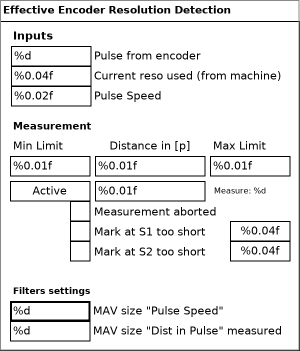
VISUALIZATION _VISU_EffectiveEncoderResolutionDetection  // 300x351
VAR_IN_OUT
	mInst : FB_EffectiveEncoderResolutionDetection;
END_VAR
    Rectangle (0,21 300x330)
    Rectangle (10,116 80x20), "Measurement"
    RoundedRectangle (10,181 80x20), "Active", colour toggle: mInst.bMeasurementActive
    Rectangle (95,156 110x20), "%0.01f", text variable: mInst.fDisInPulse
    Rectangle (95,136 110x20), "Distance in [p]"
    Rectangle (91,86 200x20), "Pulse Speed"
    Rectangle (11,86 80x20), "%0.02f", text variable: mInst.fSpeed
    Rectangle (91,46 200x20), "Pulse from encoder"
    Rectangle (11,46 80x20), "%d", text variable: mInst.nPulse
    Rectangle (11,66 80x20), "%0.04f", text variable: mInst.fCurrentResolution, input disabled if: TRUE
    Rectangle (91,66 200x20), "Current reso used (from machine)"
    Rectangle (10,281 80x20), "Filters settings"
    Rectangle (90,301 200x20), "MAV size "Pulse Speed""
    Rectangle (90,321 200x20), "MAV size "Dist in Pulse" measured"
    Rectangle (10,321 80x20), "%d", text variable: mInst.nDisInPulseFilterSz, input disabled if: TRUE
    Rectangle (10,26 80x20), "Inputs"
    Rectangle (0,0 240x20), "Effective Encoder Resolution Detection"
    Rectangle (211,181 80x20), "Measure: %d", tooltip "measurement counter", text variable: mInst.nMeasurementCounter
    Rectangle (10,156 80x20), "%0.01f", tooltip "Limits from machine", text variable: mInst.fEncoderPulseDistMin, colour toggle: mInst.bLower, input disabled if: TRUE
    Rectangle (210,156 80x20), "%0.01f", tooltip "Limits from machine", text variable: mInst.fEncoderPulseDistMax, colour toggle: mInst.bHigher, input disabled if: TRUE
    Rectangle (10,136 80x20), "Min Limit"
    Rectangle (210,136 80x20), "Max Limit"
    RoundedRectangle (70,201 20x20), colour toggle: mInst.bAborted
    Rectangle (91,202 200x20), "Measurement aborted"
    RoundedRectangle (70,221 20x20), colour toggle: mInst.bMarkTooShort_S1
    Rectangle (91,222 200x20), "Mark at S1 too short"
    RoundedRectangle (70,241 20x20), colour toggle: mInst.bMarkTooShort_S2
    Rectangle (91,242 200x20), "Mark at S2 too short"
    Rectangle (230,221 60x20), "%0.04f", tooltip "Mark length in [mm], minimum length=%0.02f [mm]", text variable: mInst.nMarkLength_S1/1000, colour toggle: mInst.bMarkTooShort_S1
        p4168582468: mInst.nC_MinMarkLength/1000
    Rectangle (230,241 60x20), "%0.04f", tooltip "Mark length in [mm], minimum length=%0.02f [mm]", text variable: mInst.nMarkLength_S2/1000, colour toggle: mInst.bMarkTooShort_S2
        p4168582468: mInst.nC_MinMarkLength/1000
    Rectangle (95,181 110x20), "%0.01f", text variable: mInst.nCurrentDistActive
    Rectangle (10,301 80x20), "%d", text variable: mInst.nSpeedFilterSz
END_VISUALIZATION

(* stored: Version 1.1.0.1, ProductVersion 3.1.4024.11
   Visu _VISU_EffectiveEncoderResolutionDetection: Id {93cc7bee-2aac-448b-bf4c-7f70cfc2d34a} *)
